PROGRAM prg_ThermostaatregelingTijdsturing
VAR
	
END_VAR

END_PROGRAM

(* stored: Version 1.1.0.1, ProductVersion 3.1.4026.12
   POU prg_ThermostaatregelingTijdsturing: Id {2d87b2cd-fdc6-4437-aac8-4dcd339217b6}, SpecialFunc None *)
